INTERFACE PUBLIC AbortingCommands EXTENDS ActionStateCommands

END_INTERFACE

(* stored: Version 1.1.0.1, ProductVersion 3.1.4026.18
   Itf AbortingCommands: Id {d9a12bf1-10a0-0e97-0748-591bd5c252aa} *)
